Staubli VAL3: OnEvent2.pgx

program OnEvent2()
  local bool l_bRes
begin
  //-----------------------------------------------------------------------
  //Header begin
  //LasMAN3.7
  //Description of program
  //
  //Input parameters
  //
  //Output paramaters
  //Example
  //  call OnEvent1()
  //History
  //  Creation : 2013-06-23  y.ye@staubli.com
  //Header end
  //-----------------------------------------------------------------------
  DataBase:bStopPoll=true
  call TxtFile:ReadCfg(l_bRes)
  IO:bWeldEnable=TxtFile:bWeldEnable
  DataBase:bStopPoll=false
  if l_bRes
    call Kit:Align(TxtFile:tCfg)
  else
    popUpMsg("读取配置文件出错")
  endIf
  DataBase:nInterfaceType=9
end
